PROGRAM Prg_Loops
VAR
	Buttons: ARRAY[1..4] OF BOOL;
	AnalogSensor: ARRAY[1..4] OF INT := [5, 6, 7, 8];
	Coils: ARRAY[1..4] OF BOOL;
	
	i: INT;
END_VAR

FOR i:=1 TO 4 BY 1 DO
	IF Buttons[i] = TRUE AND AnalogSensor[i] > 6 THEN
		Coils[i]:=TRUE;
	ELSE
		Coils[i]:=FALSE;
	END_IF
END_FOR

END_PROGRAM

(* stored: Version 1.1.0.1, ProductVersion 3.1.4024.9
   POU Prg_Loops: Id {29c32d61-f63f-4d2f-b732-aeb08558828a}, SpecialFunc None *)
